Fanuc KAREL source: f_hand_t.kl

PROGRAM F_HAND_T
BEGIN
    CLOSE HAND 1
    RELAX HAND 2
    OPEN HAND 5
END F_HAND_T
